Universal Robots URScript: string_waypoints.script

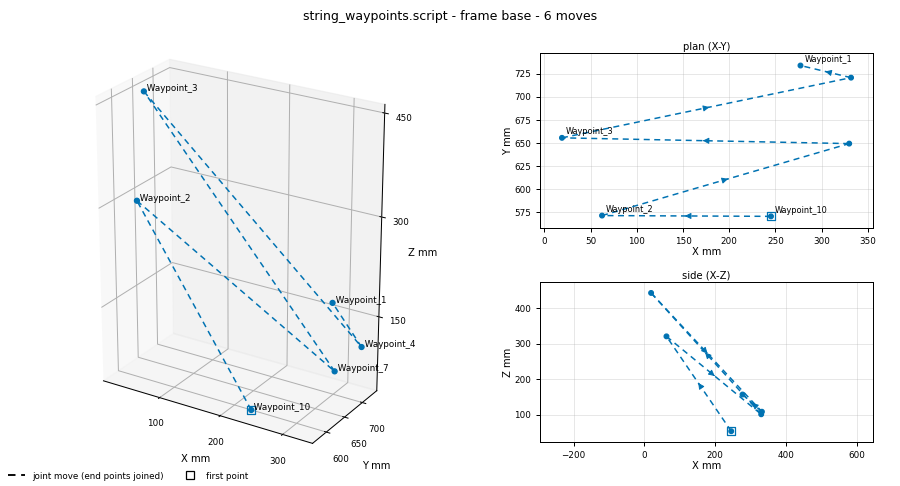
[picture p0: tool path of string_waypoints.script in frame base, 6 of 6 moves have a stored position in this frame; points joined in program order, loops and branches not executed]
def unnamed():
  global _hidden_verificationVariable=0
  step_count_bb5a21a6_9985_464d_b23e_3d0750e3f764 = 0.0
  thread Step_Counter_Thread_eaaca717_f518_4694_a4f2_ed4869ce81b8():
    while (True):
      step_count_bb5a21a6_9985_464d_b23e_3d0750e3f764 = step_count_bb5a21a6_9985_464d_b23e_3d0750e3f764 + 1.0
      sync()
    end
  end
  run Step_Counter_Thread_eaaca717_f518_4694_a4f2_ed4869ce81b8()
  set_gravity([0.0, 0.0, 9.82])
  set_tcp(p[0.028210348281514253,-0.09610723587300697,-0.09969041498611403,0.0,0.0,0.0])
  set_tool_communication(False, 115200, 0, 1, 1.5, 3.5)
  set_tool_output_mode(0)
  set_tool_digital_output_mode(0, 1)
  set_tool_digital_output_mode(1, 1)
  set_tool_voltage(0)
  set_safety_mode_transition_hardness(1)
  set_target_payload(0.260000, [0.050000, -0.008000, 0.024000], [0.000163, 0.000163, 0.000163, 0.000000, 0.000000, 0.000000])
  set_standard_analog_input_domain(0, 1)
  set_standard_analog_input_domain(1, 1)
  set_tool_analog_input_domain(0, 1)
  set_tool_analog_input_domain(1, 1)
  set_analog_outputdomain(0, 0)
  set_analog_outputdomain(1, 0)
  set_input_actions_to_default()
  global Plane_1=p[0.32571614183608727,0.7933870146316717,0.11820742021636722,-2.208244884171713,-0.24738609815952348,-1.9195085473101943]
  global Plane_2=p[0.3436052139151623,0.7478032414335104,0.10077839665899768,2.768545736097797,0.1284831553507919,1.3672805628273381]
  global Plane_3=p[0.31945151854627996,0.6757990361168175,0.09459088830114093,2.7301760593116526,-0.049483824131046385,1.4252239353300047]
  global Plane_4=p[0.3372257363094211,0.6222230974198586,0.07001667903587716,2.621672423508307,-0.12240385890263918,1.4373011913128484]
  # begin: URCap Installation Node
  #   Source: External Control, 1.0.5, FZI Research Center for Information Technology
  #   Type: External Control
  # end: URCap Installation Node
  global Waypoint_10_p=p[.245283703052, .570710326777, .053265630190, -1.842545665824, -1.391797994920, .068711419486]
  global Waypoint_10_q=[-2.3077740403406404, -0.4328001930296841, 1.6809992346605778, -2.955228773678524, -0.7451124352554306, -1.9653584271955937]
  global Waypoint_2_p=p[.062353052662, .571559213046, .321200952358, -1.565895790305, -1.647200942960, .323013909317]
  global Waypoint_2_q=[-2.0261486212359827, -1.0770766300014039, 1.9167802969561976, -2.4172259769835414, -0.6785553137408655, -2.0693939367877405]
  global Waypoint_7_p=p[.329981083328, .649486277860, .101065034548, -1.703295403645, -1.726838059501, .635956202439]
  global Waypoint_7_q=[-2.3168001871441124, -0.49838953498327676, 1.3082145111680712, -1.830637521466719, -0.9392310725615527, -2.5102874725149733]
  global Waypoint_3_p=p[.018957161096, .655733371797, .443884694554, -1.647651663719, -1.773345041841, .627023911463]
  global Waypoint_3_q=[-1.9138854185687464, -1.1527564090541382, 1.5585396925555628, -1.7306763134398402, -0.7847922484027308, -2.087546173726217]
  global Waypoint_4_p=p[.331972829410, .720894243842, .108291188914, -1.644956394239, -2.108101774266, 1.059071414057]
  global Waypoint_4_q=[-2.264972537227802, -0.3778790224680133, 0.914086507142451, -1.334612975905629, -1.3422730752938108, -2.6009259901948476]
  global Waypoint_1_p=p[.277236601206, .734032359319, .156891527665, 1.738924275492, 2.310428552465, -1.107753563859]
  global Waypoint_1_q=[-2.210412708052746, -0.49084595566760747, 0.9551938502229333, -1.302301742823495, -1.605072055336045, -2.4750900912233345]
  while (True):
    $ 2 "Robot Program"
    $ 3 "MoveJ"
    $ 4 "Waypoint_10" "breakAfter"
    movej(get_inverse_kin(Waypoint_10_p, qnear=Waypoint_10_q), a=1.3962634015954636, v=1.0471975511965976)
    $ 5 "Waypoint_2" "breakAfter"
    movej(get_inverse_kin(Waypoint_2_p, qnear=Waypoint_2_q), a=1.3962634015954636, v=1.0471975511965976)
    $ 6 "MoveJ"
    $ 7 "Waypoint_7" "breakAfter"
    movej(get_inverse_kin(Waypoint_7_p, qnear=Waypoint_7_q), a=1.3962634015954636, v=1.0471975511965976)
    $ 8 "Waypoint_3" "breakAfter"
    movej(get_inverse_kin(Waypoint_3_p, qnear=Waypoint_3_q), a=1.3962634015954636, v=1.0471975511965976)
    $ 9 "MoveJ"
    $ 10 "Waypoint_4" "breakAfter"
    movej(get_inverse_kin(Waypoint_4_p, qnear=Waypoint_4_q), a=1.3962634015954636, v=1.0471975511965976)
    $ 11 "MoveJ"
    $ 12 "Waypoint_1" "breakAfter"
    movej(get_inverse_kin(Waypoint_1_p, qnear=Waypoint_1_q), a=1.3962634015954636, v=1.0471975511965976)
  end
end
